// TwinCAT 3 PLC project PLCIO
// ProgramVersion: 3.1.4026.10
// libraries:
//   Tc2_ControllerToolbox, * (Beckhoff Automation GmbH)
//   Tc2_IoFunctions, * (Beckhoff Automation GmbH)
//   Tc2_ModbusRTU, * (Beckhoff Automation GmbH)
//   Tc2_ModbusSrv, * (Beckhoff Automation GmbH)
//   Tc2_SerialCom, * (Beckhoff Automation GmbH)
//   Tc2_Standard, * (Beckhoff Automation GmbH)
//   Tc2_System, * (Beckhoff Automation GmbH)
//   Tc2_Utilities, * (Beckhoff Automation GmbH)
//   Tc3_BA_Common, * (Beckhoff Automation GmbH)
//   Tc3_EventLogger, * (Beckhoff Automation GmbH)
//   Tc3_Module, * (Beckhoff Automation GmbH)
// project tree:
//   / CheckDivDInt.TcPOU, CheckDivLInt.TcPOU (not stored), CheckDivLReal.TcPOU, CheckDivReal.TcPOU (not stored), PlcTask.TcTTO (not stored), PlcTask_Fast.TcTTO (not stored)
//   DUTs/ outWord.TcDUT, ScaleFactor.TcDUT, ST_Device.TcDUT, RecipeStep.TcDUT
//   FUNTION/ BOOL_TO_STRING_LHeaterON.TcPOU, CheckRangeSigned.TcPOU (not stored), CheckRangeUnsigned.TcPOU (not stored), HEXSTR_TO_REAL_LHeaterPV.TcPOU, Real_To_String_LineHeater.TcPOU, Real_To_String_ThermalBath.TcPOU, USINT_TO_WORD_Bit.TcPOU, WORD_TO_USINT_Bit.TcPOU (not stored)
//   GVLs/ GVL.TcGVL (not stored), GVL_Interlock.TcGVL, GVL_Serial.TcGVL (not stored), GVL_IO.TcGVL, RCP.TcGVL (not stored)
//   POUs/ FB_RecipeSequencer.TcPOU (not stored), backup2.TcPOU (not stored), backup1.TcPOU, Test_Recipe_Run.TcPOU, FB_RampGeneration_Gas.TcPOU (not stored), MAIN.TcPOU (not stored), P11_E3508.TcPOU, P12_IQ_PLUS.TcPOU, P13_LineHeater.TcPOU, P14_ThermalBath.TcPOU (not stored), P15_RotationOperation.TcPOU (not stored), P16_CoverOperation.TcPOU (not stored), P17_DOROperation.TcPOU (not stored), P20_BackgroundCom.TcPOU, P21_Background_LineHeater.TcPOU (not stored), P22_Background_ThermalBath.TcPOU (not stored), P50_RecipeControl.TcPOU (not stored), P90_Interlock.TcPOU (not stored), P91_Monitoring.TcPOU (not stored), P92_Maintenance.TcPOU (not stored), P93_Setting.TcPOU (not stored)

// ---- DUTs/outWord.TcDUT
TYPE outWord :
STRUCT
	Lower : USINT; //Lower Bytes
	Upper : USINT; //Upper Bytes
END_STRUCT
END_TYPE

// ---- DUTs/ScaleFactor.TcDUT
TYPE ScaleFactor :
STRUCT
	MinFactor	: USINT; // Sensor Minimum Range
	MaxFactor	: USINT; // Sensor Maximum Range
END_STRUCT
END_TYPE

// ---- DUTs/ST_Device.TcDUT
TYPE ST_Device :
STRUCT
	aDigitalInputIO  	: ARRAY[1..9]OF BYTE; //KL1408 9EA
	aDigitalOutputIO  	: ARRAY[1..4]OF BYTE; //KL2408 4EA
	
	// Analog Input to INT
	aAnalogInputIO 		: ARRAY[1..40]OF INT;
	aAnalogOutputIO 	: ARRAY[1..28]OF INT;
	aAnalogInputIO2 	: ARRAY[1..2]OF UINT;
	//Solenoid Valve
	aOutputSolValve  	: ARRAY[1..2]OF DWORD; //Solenoid Valve 
END_STRUCT
END_TYPE

// ---- DUTs/RecipeStep.TcDUT
TYPE RecipeStep :
STRUCT
	iRecipe : ARRAY[1..9] OF INT; //Reactor Condition
	rRecipe : ARRAY[1..26] OF REAL; //MFC, EPC Data
	dRecipe : DWORD; //Valve Data
	sRecipe : STRING(81);
END_STRUCT
END_TYPE

// ---- GVLs/GVL_Interlock.TcGVL
{attribute 'qualified_only'}
VAR_GLOBAL
	
END_VAR

// ---- GVLs/GVL_IO.TcGVL
{attribute 'qualified_only'}
VAR_GLOBAL
	// Digital IO to Byte
	aDigitalInputIO AT %I* 	: ARRAY[1..9]OF BYTE; //KL1408 9EA
	aDigitalOutputIO AT %Q* : ARRAY[1..4]OF BYTE; //KL2408 4EA

	// Analog Input to INT
	aAnalogInputIO AT %I* 	: ARRAY[1..40]OF INT;
	aAnalogOutputIO AT %Q* 	: ARRAY[1..28]OF INT;
	aAnalogInputIO2 AT %I*	: ARRAY[1..2]OF UINT;
	//Solenoid Valve
	aOutputSolValve AT %Q* 	: ARRAY[1..2]OF DWORD; //Solenoid Valve 
	// Variable(struct) Connecting PC to PLC 
	stDeviceIO				: ST_Device;

	aMaxValue	: ARRAY[1..50]OF REAL; //Device Max Value from UI
	
	
END_VAR

// ---- CheckDivDInt.TcPOU
// Implicitly generated code : DO NOT EDIT
FUNCTION CheckDivDInt : DINT
VAR_INPUT
	divisor:DINT;
END_VAR

// Implicitly generated code: Only an implementation suggestion
{noflow}
IF divisor = 0 THEN
	CheckDivDInt:=1;
ELSE
	CheckDivDInt:=divisor;
END_IF;

END_FUNCTION

// ---- CheckDivLReal.TcPOU
// Implicitly generated code : DO NOT EDIT
FUNCTION CheckDivLReal : LREAL
VAR_INPUT
	divisor:LREAL;
END_VAR

// Implicitly generated code: Only an implementation suggestion
{noflow}
IF divisor = 0 THEN
	CheckDivLReal:=1;
ELSE
	CheckDivLReal:=divisor;
END_IF;

END_FUNCTION

// ---- FUNTION/BOOL_TO_STRING_LHeaterON.TcPOU
FUNCTION BOOL_TO_STRING_LHeaterON : STRING
VAR_INPUT
	nHeaterNumber	: INT;
	bON				: BOOL;
END_VAR
VAR
	sString			: STRING;
	sHeaterNumber	: STRING;
END_VAR

//LH: Line Heater x 8EA -> 8Channel TIC 1EA
//Model: HANYOUNG NUX, MC9-8RD0SS32

//STRING : '$0201DWR,02,0302(CH_NO),0001(CH_1),0501(AT),0001(AT-ON)
sString := '$0201DWR,02,0302,,0501,000$0D$0A';

//Convert to Channel from Heater Number
sHeaterNumber := DINT_TO_DECSTR(nHeaterNumber, 4);
sString := INSERT(sString,sHeaterNumber,15);

IF bON = TRUE THEN
	sString := INSERT(sString,'1',28);
ELSE
	sString := INSERT(sString,'0',28);
END_IF

BOOL_TO_STRING_LHeaterON := sString;

END_FUNCTION

// ---- FUNTION/HEXSTR_TO_REAL_LHeaterPV.TcPOU
FUNCTION HEXSTR_TO_REAL_LHeaterPV : REAL
VAR_INPUT
	hStrTemperaturePV : STRING;
END_VAR
VAR
	hData			:UDINT;
	aData	: ARRAY[0..1]OF BYTE;
	bSwap	: BYTE;
	ptStrTemperature : POINTER TO INT;
	nTemperaturePV : INT;
END_VAR

// Convert to Data Array from HexString
hData := HEXSTR_TO_DATA(hStrTemperaturePV, ADR(aData), SIZEOF(aData));

//Swap Data
bSwap := aData[0];
aData[0] := aData[1];
aData[1] := bSwap;

ptStrTemperature := ADR(aData);
nTemperaturePV := ptStrTemperature^;
HEXSTR_TO_REAL_LHeaterPV := INT_TO_REAL(nTemperaturePV);

END_FUNCTION

// ---- FUNTION/Real_To_String_LineHeater.TcPOU
FUNCTION Real_To_String_LineHeater : STRING
VAR_INPUT
	rTemperatureSV 		: REAL;
	nHeaterNumber		: INT;
END_VAR
VAR
	wTemperature		: WORD;
	hStrTemp			: STRING;
	sHeaterNumber		: STRING;
	sString				: STRING;
	sSendString			: STRING;
END_VAR

//LH: Line Heater x 8EA -> 8Channel TIC 1EA
//Model: HANYOUNG NUX, MC9-8RD0SS32

// Multiple decimal place point
// STRING : '$0201DWR,03,0301(ZONE_NO),0001(ZONE_1),0302(CH_NO),0001(CH_1,sHeaterNumber),0401(SV), hStrTemp, $0D$0A'
sString := '$0201DWR,03,0301,0001,0302,,0401,,$0D$0A';

//Convert to Channel from Heater Number
sHeaterNumber := DINT_TO_DECSTR(nHeaterNumber, 4);
sString := INSERT(sString,sHeaterNumber,25);
	
//Convert to String Type
wTemperature := REAL_TO_WORD(rTemperatureSV);
hStrTemp := WORD_TO_HEXSTR(wTemperature, 4, FALSE);
Real_To_String_LineHeater := INSERT(sString,hStrTemp,35);

END_FUNCTION

// ---- FUNTION/Real_To_String_ThermalBath.TcPOU
FUNCTION Real_To_String_ThermalBath : STRING
VAR_INPUT
	rTemperatureSV 	: REAL;
	nBathNumber		: INT;
END_VAR
VAR
	sBathNumber 	: STRING;
	rTemp 			: REAL;
	nTemp 			: DINT;
	sTemp 			: STRING;
	sBaseString		: STRING;
END_VAR

// Thermal Bath SMC HEBC002-WA10
rTemp := rTemperatureSV*10 ;
nTemp := REAL_TO_DINT(rTemp);
sBaseString := '$020WSV1$03';

sBathNumber := INT_TO_STRING(nBathNumber);
sBaseString := INSERT(sBaseString,sBathNumber,2);

IF nTemp >= 0 THEN
	sTemp := DINT_TO_DECSTR(nTemp, 5); //00010
ELSE
	sTemp := DINT_TO_DECSTR(nTemp, 4); 
	sTemp := CONCAT('-',sTemp); //-0010
END_IF

sBaseString := INSERT(sBaseString,sTemp,7);

Real_To_String_ThermalBath := sBaseString;

END_FUNCTION

// ---- FUNTION/USINT_TO_WORD_Bit.TcPOU
//2-USINT combine to 1-WORD converting using a bit operation
FUNCTION USINT_TO_WORD_Bit : WORD
VAR_INPUT
	aInput_L : USINT; //Lower
	aInput_U : USINT; //Upper
END_VAR
VAR
	nWord_L : WORD; //Lower
	nWord_U : WORD; //Upper
END_VAR

nWord_L := TO_WORD(aInput_L);
// 1111_1111
// 0000_0000_1111_1111
nWord_U := TO_WORD(aInput_U);
// 1111_1111
// 0000_0000_1111_1111
nWord_U := SHL(nWord_U, 8);
// 1111_1111_0000_0000
USINT_TO_WORD_Bit := TO_WORD(nWord_L OR nWord_U);

END_FUNCTION

// ---- POUs/backup1.TcPOU
PROGRAM P50_RecipeControl1
VAR
	RcpIndex	: INT;
	
	iTimerCount: INT;
	OnTimer: TON;
	OffTimerOut: BOOL;
	OnTimerOut: BOOL;
	timeTrigOn: R_TRIG;
	
	bTrigOn: BOOL;
	ReverseSignal: BOOL;
	OffTimer: TOF;
	fb_RecipeSequencer : FB_RecipeSequencer;
END_VAR

IF RCP.bRcpInit THEN
	(* reset the init flag *)
	iTimerCount := 0;
	RcpIndex := 1;
	RCP.bRcpInit := FALSE;
END_IF

IF RcpIndex <= RCP.iRcpTotalStep THEN
	OnTimer(IN:=OffTimerOut, Pt:= INT_TO_TIME(500), Q=>OnTimerOut, ET=>);
	timeTrigOn(clk:=OnTimerout, Q=>bTrigOn);
	IF (bTrigOn AND RCP.iRcpOperationState) THEN
		iTimerCount := iTimerCount +1;
		bTrigOn := FALSE;
		
		IF iTimerCount <= RCP.aRecipe[RcpIndex].iRecipe[2] THEN
			fb_RecipeSequencer(nRcpIndex:=RcpIndex);
			
		ELSIF iTimerCount > RCP.aRecipe[RcpIndex].iRecipe[2] + RCP.aRecipe[RcpIndex].iRecipe[3] THEN
			iTimerCount := 0;
			RcpIndex := RcpIndex + 1;
		END_IF
	END_IF
	IF OnTimerOut = TRUE THEN
		ReverseSignal := FALSE;
	ELSE
		ReverseSignal := TRUE;
	END_IF

	OffTimer(in:=ReverseSignal, pt:= INT_TO_TIME(500), q=>OffTimerOut,et=>);
END_IF

END_PROGRAM

// ---- POUs/Test_Recipe_Run.TcPOU
PROGRAM Test_Recipe_Run
VAR
// 	fb_RecipeSequencer : FB_RecipeSequencer;
	bMaintKey : BOOL;
	bPc2Plc	: BOOL;
	
	plc_state	: BOOL;
	plc_array	: BYTE;
	
	iRcpCurrNum : INT := 1;
	iTimerCount	: INT;

	timeTrigOn	: r_trig;
	bTrigOn		: BOOL;
	bRcpInit	: BOOL;
	bRcpEnable	: BOOL;
	fb_RecipeSequencer : FB_RecipeSequencer;

	ctime : TIME :=  T#1D14H30M40S500MS;
	lctime : LTIME ;
	
	cdate : DATE :=  D#2024-07-07;
	str : STRING ;
	wstr : STRING;
	tempstr : STRING;

	OnTimer : TON;
	OffTimer : TOF;
	EnableTimer : BOOL;
	TimerOutPut : BOOL;	
	OnTimerOut : BOOL := FALSE;
	ReverseSignal : BOOL;
	OffTimerOut : BOOL;
	count : INT;
	el2088_out : BYTE;
	el4024_out : INT;
	el3054_in : INT;
	
END_VAR

// Load current recipe of recipes array 
bMaintKey := GVL_IO.aDigitalInputIO[1].0;

// Connect PLC varibaes to PC variables
IF bPc2Plc = TRUE THEN
	GVL_IO.aDigitalInputIO := GVL_IO.stDeviceIO.aDigitalInputIO;
	GVL_IO.aDigitalOutputIO := GVL_IO.stDeviceIO.aDigitalOutputIO;
	GVL_IO.aAnalogInputIO := GVL_IO.stDeviceIO.aAnalogInputIO;
	GVL_IO.aAnalogOutputIO := GVL_IO.stDeviceIO.aAnalogOutputIO;
	GVL_IO.aAnalogInputIO2 := GVL_IO.stDeviceIO.aAnalogInputIO2;
	GVL_IO.aOutputSolValve := GVL_IO.stDeviceIO.aOutputSolValve;
	bPc2Plc := FALSE;
ELSE
	GVL_IO.stDeviceIO.aDigitalInputIO  := GVL_IO.aDigitalInputIO; 
	GVL_IO.stDeviceIO.aDigitalOutputIO := GVL_IO.aDigitalOutputIO;
	GVL_IO.stDeviceIO.aAnalogInputIO   := GVL_IO.aAnalogInputIO;
	GVL_IO.stDeviceIO.aAnalogOutputIO  := GVL_IO.aAnalogOutputIO; 
	GVL_IO.stDeviceIO.aAnalogInputIO2  := GVL_IO.aAnalogInputIO2; 
	GVL_IO.stDeviceIO.aOutputSolValve  := GVL_IO.aOutputSolValve;
END_IF

IF bRcpInit THEN
	(* reset the init flag *)
	iTimerCount := 0;
	iRcpCurrNum := 1;
	bRcpInit := FALSE;
END_IF

IF iRcpCurrNum <= 50 THEN
	OnTimer(IN:=OffTimerOut, Pt:= INT_TO_TIME(500), Q=>OnTimerOut, ET=>);
	timeTrigOn(clk:=OnTimerout, Q=>bTrigOn);
	IF (bTrigOn AND GVL.bRunRecipe) THEN
		iTimerCount := iTimerCount +1;
		bTrigOn := FALSE;
		
		IF iTimerCount <= RCP.aRecipe[iRcpCurrNum].iRecipe[2] THEN
			fb_RecipeSequencer(nRcpIndex:=iRcpCurrNum);
			
		ELSIF iTimerCount > RCP.aRecipe[iRcpCurrNum].iRecipe[2] + RCP.aRecipe[iRcpCurrNum].iRecipe[3] THEN
			iTimerCount := 0;
			iRcpCurrNum := iRcpCurrNum + 1;
		END_IF
	END_IF
	IF OnTimerOut = TRUE THEN
		ReverseSignal := FALSE;
	ELSE
		ReverseSignal := TRUE;
	END_IF

	OffTimer(in:=ReverseSignal, pt:= INT_TO_TIME(500), q=>OffTimerOut,et=>);
END_IF


cdate :=  D#2024-07-07;
str := 'We are the one, let us heading forwards';

count := count + 1;

GVL.EL4024_OUT := el4024_out;
el3054_in := GVL.EL3054_IN;

plc_array := EL2088_OUT;

END_PROGRAM

// ---- POUs/P11_E3508.TcPOU
PROGRAM P11_E3508
VAR_INPUT
	nTemperatureTargetValue	: INT(0..1200); //Target Values, Input Range 0 ~ 1200 Celcius
	nRampTime				: INT := 1; //Second
	nPowerRateSetValue		: WORD;	
	bOutputManAuto 			: BOOL; // 0:Auto, 1:Manual Operation
	
	bHeaterOn				: BOOL := FALSE; //to PSTEK
	bHeaterReset			: BOOL; //to PSTEK

END_VAR
VAR_OUTPUT
	bAlarmState_E3508 		: BOOL; //Alarm or Sensor Break Signal
	bManAuto_E3508 			: BOOL; // 0:Manual, 1:Auto
	rPowerRate				: REAL;	//Power rate for Monitoring
	
	isHeaterReady			: BOOL; //Close : Ready
	isHeaterRun				: BOOL; //Close : Running, Open : Stop
	isHeaterFault			: BOOL; //Close : Falut, Open : Normal
	//isInductionHeaterErr	: BOOL; //Power Supply
	bInductionHeaterCB		: BOOL;
END_VAR

VAR
	//Input from E3508 Controller
	aInputPVBytes AT %I* 		: ARRAY[1..2]OF USINT; //Input Process Values
	aInputSVBytes AT %I* 		: ARRAY[1..2]OF USINT; //Input Set Values
	aInputTVBytes AT %I* 		: ARRAY[1..2]OF USINT; //Input Target Valuse
	aInputCVBytes AT %I* 		: ARRAY[1..2]OF USINT; //Induction Heter Controlled Values
	aInputProportional AT %I* 	: ARRAY[1..2]OF USINT; //PID - Proportional Band
	aInputIntegral AT %I* 		: ARRAY[1..2]OF USINT; //PID - Integral Time
	aInputDerivative AT %I* 	: ARRAY[1..2]OF USINT; //PID - Derivative Time 
	nInputAlarmBytes AT %I* 	: USINT; // Alarm State
	nInputManAutoBytes AT %I* 	: USINT; // ManAuto State
	
	nTemperaturePV_E3508		: WORD;
	nTemperatureSV_E3508		: WORD;
	nPowerRate_E3508		: WORD; //To Induction Heater Control Values
	nParameterP				: WORD; //PID Parameter P
	nParameterI				: WORD; //PID Parameter I
	nParameterD				: WORD; //PID Parameter D
	//Output to E3508 Controller
	wOutputSVBytes 				: outWord;
	wOutputPowerSVBytes 		: outWord;
	aOutputSVBytes AT %Q* 		: ARRAY[1..2]OF USINT; //Temperature Set Value
	nOutputManAutoBytes AT %Q* 	: USINT; //ManAuto Change
	aOutputPowerBytes AT %Q* 	: ARRAY[1..2]OF USINT; //Output Power in Manual State
	//nOutputAlarmClear AT %Q* : USINT; //Alarm Clear Set
	
	nTemperatureControlValue	: WORD;
	
	// for FB_CTRL_RAMP_GENERATOR Variable
	(* input *)
	bEnable					: BOOL;
	rTemperatureStartValue	: REAL;
	rTemperatureTargetValue	: REAL;
	(* output *)
	rTemperatureControlValue : LREAL;
	bValueReached			: BOOL;
	(* function block *)
	fbCTRL_RAMP_GENERATOR		: FB_CTRL_RAMP_GENERATOR;
	stCTRL_RAMP_GENERATOR_PARAMS: ST_CTRL_RAMP_GENERATOR_PARAMS;

	eErrorId				: E_CTRL_ERRORCODES;
	bError					: BOOL;
	bInit					: BOOL := TRUE;

	(* Induction Heating Operation Parameter*)
	rRampingRatio			: REAL;	
END_VAR

//Induction Heater & Temperature Controller & Thermo Couple(R-Type)
//Maker: PSTEK, Eurotherm
//Model: 3508
//Temperature Range: 0 ~ 12000℃

(* Read from Power Distribution Pannel *)
bInductionHeaterCB		:= GVL_IO.aDigitalInputIO[4].7;

(* Read from E3508 Device Value *)
nTemperaturePV_E3508	:= USINT_TO_WORD_Bit(aInputPVBytes[1], aInputPVBytes[2]);
nTemperatureSV_E3508	:= USINT_TO_WORD_Bit(aInputSVBytes[1], aInputSVBytes[2]);
nPowerRate_E3508		:= USINT_TO_WORD_Bit(aInputCVBytes[1], aInputCVBytes[2]); //divided to 10
nParameterP 			:= USINT_TO_WORD_Bit(aInputProportional[1], aInputProportional[2]);
nParameterI 			:= USINT_TO_WORD_Bit(aInputIntegral[1], aInputIntegral[2]);
nParameterD 			:= USINT_TO_WORD_Bit(aInputDerivative[1], aInputDerivative[2]);

bAlarmState_E3508 		:= nInputAlarmBytes.7;
bManAuto_E3508 			:= nInputManAutoBytes.7;

(* Read from Induction Heater Value *)
isHeaterReady 			:= GVL_IO.aDigitalInputIO[2].2;
isHeaterRun		 		:= GVL_IO.aDigitalInputIO[2].3;
isHeaterFault 			:= GVL_IO.aDigitalInputIO[2].4;

(*Ramp Generator Parameter Variable*)
rTemperatureTargetValue	:= INT_TO_REAL(nTemperatureTargetValue);
rPowerRate				:= WORD_TO_REAL(nPowerRate_E3508)*0.1; //divided to 10

bHeaterOn := TRUE;
bInit := NOT((rTemperatureTargetValue = 0) AND (rTemperatureStartValue = 0));

IF bInit AND nRampTime <> 0 AND RCP.iRcpOperationState=10 THEN
	rRampingRatio := ABS(rTemperatureTargetValue - rTemperatureStartValue) / nRampTime; //Second
	(* init parameter struct *)
	stCTRL_RAMP_GENERATOR_PARAMS.tTaskCycleTime		:= T#2MS;
	stCTRL_RAMP_GENERATOR_PARAMS.tCtrlCycleTime		:= T#100MS;
	stCTRL_RAMP_GENERATOR_PARAMS.fVeloPos			:= rRampingRatio; (* in units per second *)
	stCTRL_RAMP_GENERATOR_PARAMS.fVeloNeg			:= rRampingRatio; (* in units per second *)

	IF rTemperatureTargetValue <> rTemperatureStartValue THEN
		bEnable := TRUE;
		(* call function block *)
		fbCTRL_RAMP_GENERATOR(
			bEnable			:= bEnable,
			fStart			:= rTemperatureStartValue,
			fTarget			:= rTemperatureTargetValue,
			stParams		:= stCTRL_RAMP_GENERATOR_PARAMS,
			fOut			=> rTemperatureControlValue,
			bValueReached	=> bValueReached,
			bError			=> bError,
			eErrorId		=> eErrorId);
	ELSE
		fbCTRL_RAMP_GENERATOR.bEnable := FALSE;
	END_IF

	IF bValueReached THEN
		rTemperatureStartValue	:= LREAL_TO_REAL(rTemperatureControlValue);
	END_IF
END_IF

nTemperatureControlValue	:= LREAL_TO_WORD(rTemperatureControlValue);

(* Write to E3508 Device Value *)
wOutputSVBytes 			:= WORD_TO_USINT_Bit(nTemperatureControlValue);
aOutputSVBytes[1] 		:= wOutputSVBytes.Lower;
aOutputSVBytes[2] 		:= wOutputSVBytes.Upper;

// PowerRate Operation
nOutputManAutoBytes.0 	:= bOutputManAuto;

wOutputPowerSVBytes 	:= WORD_TO_USINT_Bit(nPowerRateSetValue*10); //multiple to 10
aOutputPowerBytes[1] 	:= wOutputPowerSVBytes.Lower;
aOutputPowerBytes[2] 	:= wOutputPowerSVBytes.Upper;

(* Write to Induction Heater Value *)
GVL_IO.aDigitalOutputIO[2].0 := bHeaterOn;
GVL_IO.aDigitalOutputIO[2].1 := bHeaterReset;

END_PROGRAM

// ---- POUs/P12_IQ_PLUS.TcPOU
PROGRAM P12_IQ_PLUS
VAR_INPUT
	nPressureTargetValue : WORD := 760;//Pressure Set Value
	nRampTime			: INT := 1; //Second
	//wSetPoint 			: WORD; //Set Point
	nSetType 			: USINT; //1:Pressure Conrol, 2:Position Control
	nTValveMode 		: USINT := 0; //Valve Mode
	bPumpOn				: BOOL;
	bPumpReset			: BOOL;
	
	bEnable				: BOOL; //Value Change

END_VAR
VAR_OUTPUT
	rPressurePV_CD1 	: REAL; //CD2 Current Pressure
	rPressurePV_CD2 	: REAL; //CD2 Current Pressure
	rValvePosition 		: REAL; //Valve Position
	bVacuumPumpCB		: BOOL;
	bThrottleValveCP	: BOOL;
	nPressureControlValue	: INT;

	//nInputStatus
	ingPressureControl 	: BOOL;
	ingPositionControl 	: BOOL;
	isValveOpen 			: BOOL;
	isValveNotInitialized 	: BOOL;	
	isValveClosed 			: BOOL;
	isValveFaultState 		: BOOL;
	ingValveInitializing 	: BOOL;
	ingHoldState 			: BOOL;
	
	// Vacuum Pump Status
	isPumpFault				: BOOL;
	isPumpWarning			: BOOL;
	isPumpAlarm				: BOOL;
	isFBRunning				: BOOL;
	isPumpRunning			: BOOL;
	
END_VAR
VAR
	//Input from IQ-PLUS Throttle Valve
	nInputStatus AT %I* : USINT; //Input Status Bytes
	aInputPressurePV_CDG1 AT %I* : ARRAY[1..2]OF USINT; //CDG1 Pressure
	aInputPressurePV_CDG2 AT %I* : ARRAY[1..2]OF USINT; //CDG2 Pressure
	aInputPressureSP AT %I* : ARRAY[1..2]OF USINT; //Set Point Pressure
	aInputValvePosionPV AT %I* : ARRAY[1..2]OF USINT; //Current Valve Position
	
	wOutputSetPoint : WORD;
	oSetPoint : outWord; //Word to Byte variable
	
	//Output to IQ-PLUS Throttle Valve
	nOutputMode AT %Q* : USINT;
	aOutputSPBytes AT %Q* : ARRAY[1..2]OF USINT; //Set Pressure
	nOutputSetType AT %Q* : USINT; //1:Pressure Control, 2:Valve Position Control
	wInputPressurePV_CDG1 : WORD; //CDG1 Current Pressure, Not Used
	wInputPressurePV_CDG2 : WORD; //CDG2 Current Pressure
	wInputValvePosition : WORD; //Current Valve Position (0~100%)
	nInputStatusOld : USINT := 9; //Value Change Monitoring, First Temp value
	
	// for FB_CTRL_RAMP_GENERATOR Variable
	(* input *)
	rPressureTargetValue 		: REAL;
	rPressureStartValue 		: REAL := 760;
	(* output *)
	rPressureControlValue		: LREAL;
	bValueReached				: BOOL;
	(* function block *)
	fbCTRL_RAMP_GENERATOR			: FB_CTRL_RAMP_GENERATOR;
	stCTRL_RAMP_GENERATOR_PARAMS	: ST_CTRL_RAMP_GENERATOR_PARAMS;
	eErrorId						: E_CTRL_ERRORCODES;
	bError							: BOOL;
	bInit						: BOOL := TRUE;	
	(* Operation Parameter*)
	rRampingRatio				: REAL;	
	rPressureControlValue_torr	: lreal;
END_VAR
VAR CONSTANT
	//Conversion Parameter
	SetPointFactor : REAL := 327.67; //Range 0~7FFFh
	PressureFactor : REAL := 24.576;	//Range 0~6000h
END_VAR

//Model : IQ Plus 
//Pressure Range : 0 ~ 1,000 Torr

(* Read from Power Distribution Pannel *)
bVacuumPumpCB		:= GVL_IO.aDigitalInputIO[5].1;
bThrottleValveCP 	:= GVL_IO.aDigitalInputIO[5].5; //Throttle Valve CP

(* Read from Vacuum Pump *)
isPumpFault			:= GVL_IO.aDigitalInputIO[2].7;
isPumpWarning		:= GVL_IO.aDigitalInputIO[3].0;
isPumpAlarm			:= GVL_IO.aDigitalInputIO[3].1;
isFBRunning			:= GVL_IO.aDigitalInputIO[3].2;
isPumpRunning		:= GVL_IO.aDigitalInputIO[3].3;

(* Read from Device Value *)
// 2USINT to WORD
wInputPressurePV_CDG1 	:= USINT_TO_WORD_Bit(aInputPressurePV_CDG1[1],aInputPressurePV_CDG1[2]);
wInputPressurePV_CDG2 	:= USINT_TO_WORD_Bit(aInputPressurePV_CDG2[1],aInputPressurePV_CDG2[2]);
wInputValvePosition 	:= USINT_TO_WORD_Bit(aInputValvePosionPV[1], aInputValvePosionPV[2]);

//From IQ Plus
rPressurePV_CD1 := WORD_TO_REAL(wInputPressurePV_CDG1)/PressureFactor;
rPressurePV_CD2 := WORD_TO_REAL(wInputPressurePV_CDG2)/PressureFactor;
rValvePosition := WORD_TO_REAL(wInputValvePosition)/SetPointFactor;

nSetType := 1;
//To IQ Plus
IF nTValveMode = 0 AND nSetType = 1 THEN
	rPressureTargetValue := nPressureTargetValue * SetPointFactor * 0.1; //Pressure Control
ELSIF nTValveMode = 0 AND nSetType = 2 THEN
	rPressureTargetValue := nPressureTargetValue * SetPointFactor; // Position Control
END_IF

//Ramp Generator
bInit := NOT((rPressureTargetValue = 0) AND (rPressureStartValue = 0));

IF bInit AND nRampTime <> 0 AND RCP.iRcpOperationState=10 THEN
	rRampingRatio := ABS(rPressureTargetValue - rPressureStartValue) / nRampTime; // Second
	(* init parameter struct *)
	stCTRL_RAMP_GENERATOR_PARAMS.tTaskCycleTime		:= T#2MS;
	stCTRL_RAMP_GENERATOR_PARAMS.tCtrlCycleTime		:= T#100MS;
	stCTRL_RAMP_GENERATOR_PARAMS.fVeloPos			:= rRampingRatio; (* in units per second *)
	stCTRL_RAMP_GENERATOR_PARAMS.fVeloNeg			:= rRampingRatio; (* in units per second *)
	(* reset the init flag *)
	bInit := FALSE;

	IF rPressureTargetValue <> rPressureStartValue THEN
		bEnable := TRUE;
		(* call function block *)
		fbCTRL_RAMP_GENERATOR(
			bEnable			:= bEnable,
			fStart			:= rPressureStartValue,
			fTarget			:= rPressureTargetValue,
			stParams		:= stCTRL_RAMP_GENERATOR_PARAMS,
			fOut			=> rPressureControlValue,
			bValueReached	=> bValueReached,
			bError			=> bError,
			eErrorId		=> eErrorId);
	ELSE
		fbCTRL_RAMP_GENERATOR.bEnable := FALSE;
	END_IF

	IF bValueReached THEN
		rPressureStartValue := LREAL_TO_REAL(rPressureControlValue);
	END_IF
END_IF


wOutputSetPoint := LREAL_TO_WORD(rPressureControlValue);
oSetPoint := WORD_TO_USINT_Bit(wOutputSetPoint);
aOutputSPBytes[1] := oSetPoint.Lower;
aOutputSPBytes[2] := oSetPoint.Upper;

nOutputSetType := nSetType;

//Valve Status Initailize
IF nInputStatus <> nInputStatusOld THEN
	// Staus Initializing
	ingPressureControl := FALSE;
	ingPositionControl := FALSE;
	isValveOpen := FALSE;
	isValveNotInitialized := FALSE;	
	isValveClosed := FALSE;
	isValveFaultState := FALSE;
	ingValveInitializing := FALSE;
	ingHoldState := FALSE;
	// Status Update	
	nInputStatusOld := nInputStatus;
END_IF

//Update Valve Status
CASE nInputStatus OF
	0 : ingPressureControl := TRUE; //Pressure Control Performing.
	1 : ingPositionControl := TRUE; //Position Control Performing.	
	2 : isValveOpen := TRUE; //Valve Open, Stopped, Not Controlling.
	3 : isValveNotInitialized := TRUE; //Valve not initialized power on or RESET Command.
	4 : isValveClosed := TRUE; //Valve Closed, Stopped, Not Controlling.
	5 : isValveFaultState := TRUE; //Has faulted during valve initialization or operation.
	6 : ingValveInitializing := TRUE; //Initailizing Process.
	8 : ingHoldState := TRUE; //intermediate position, not at open or close and not controlling pressure.
END_CASE

// nOutputMode
// 0 : uses setpoint and setpoint type to control the valve.
// 1 : Does not use setpoint and setpoint type to operate the valve.
// 2 : Does not use setpoint and setpoint type to operate the valve.
// 3 : Holds valve in current position.
// 4 : Reset the controller.
nOutputMode := nTValveMode;
nPressureControlValue := LREAL_TO_INT(rPressureControlValue);

rPressureControlValue_torr := LREAL_TO_REAL(rPressureControlValue / SetPointFactor * 10);

 //Pressure Control

GVL_IO.aDigitalOutputIO[2].2 := bPumpOn; //Pump On
GVL_IO.aDigitalOutputIO[2].3 := bPumpReset; // Pump Reset

END_PROGRAM

// ---- POUs/P13_LineHeater.TcPOU
PROGRAM P13_LineHeater
VAR_INPUT
	rTemperatureSV 		: ARRAY[1..8]OF REAL;
	bAutoTuneSV 		: ARRAY[1..8]OF BOOL;
END_VAR
VAR_OUTPUT
	rTemperaturePV 		: ARRAY[1..8]OF REAL;
	isLineHeater_Run	: ARRAY[1..8]OF BOOL;
	isLineHeater_ATune	: ARRAY[1..8]OF BOOL;
	isLineHeater_Err	: ARRAY[1..8]OF BOOL;
END_VAR
VAR
	TimeOnDelay			: TON; //Time delay after Power ON of Thermal Bath
	TimeCycle			: TON;
	nComMode 			: INT; // //1 = PV Req, 2 = STATUS Req, 3 = SV Write, 4 = AutoTune On/Off
	nCount 				: INT;
	rTemperatureTV 		: ARRAY[1..8]OF REAL;
	bAutoTuneTV			: ARRAY[1..8]OF BOOL;

	//for sending variable
	TimeWaitSend		: TON;
	bSendingEnable 		: BOOL:=TRUE; // Check the Sending Stage
	bSetValueMode 		: BOOL;
	fbSend				: SendString;
	sSendString 		: STRING;
	bSendBusy			: BOOL;
	bSendingOK 			: BOOL; //v1
	eSendErrorID		: ComError_t;
	
	// for received variable
	TimeWaitReceive		:TON;
	fbReceive			: ReceiveString;
	sReceivedString		: STRING;
	bStringReceived		: BOOL;
	bReceiveBusy		: BOOL;
	bReceiveError		: BOOL;
	eReceiveErrorID		: ComError_t;
	bReceiveTimeout		: BOOL;
	bReceivedOK 		: BOOL;
	hStrReceivedST		: STRING;
	hStrReceivedPV		: STRING;
	
	nHeaterNumber 		: INT := 1;
	sHeaterNumber 		: STRING := '1';
	sReceivedHeaterNumber : STRING;
	nReceivedHeaterNumber : INT;
	sReceivedAffirmation : STRING;
	sReceivedData 		: STRING;
	nHeaterStrPositionPV : INT:= 11; //Received String Start Position
	nDecimal			:INT;
	nSendStrCounter		:INT := 1;
	bReset : BOOL;
	sTest : STRING;
	nStrPosition : INT;
	nHeaterNumberPV : INT;
	sTemperaturePV : STRING;
	(* Input *)
	bLineHeaterCB		: BOOL;
	bLineHeaterCP		: BYTE;
END_VAR

//LH: Line Heater x 8EA -> 8Channel TIC 1EA
//Maker: HANYOUNG NUX
//Model: MC9-8RD0SS32
//Temp Range: -15 ~200℃
//RS485: 9600, DataBit(8), Parity(None), StopBit(1)
//BCC Check X

(* Read from Device Value *)
// Line Heater CP
bLineHeaterCB	:= GVL_IO.aDigitalInputIO[5].2;
bLineHeaterCP 	:= GVL_IO.aDigitalInputIO[6]; //LineHeaterCP1   := bLineHeaterCP.0, Until CP8

// make a sending string
TimeOnDelay(IN:= P90_Interlock.bLineHeaterMC, PT :=T#5S); //Time Delay after a Thermal Bath MC ON
IF TimeOnDelay.Q THEN
	TimeOnDelay(IN:=FALSE);
	// Make a sending string Set value or Request value 
	IF bSendingEnable = FALSE THEN
		bSendingEnable := TRUE;
		bSendingOK := FALSE;
		bReceivedOK := FALSE;
		
		IF nComMode <>1 THEN
			sSendString := '$0201DRS,08,0001$0D$0A'; //Request PV
			nComMode := 1;
		ELSE
			sSendString := '$0201DRS,08,0111$0D$0A'; //Request State
			nComMode := 2;
		END_IF
	
		FOR nHeaterNumber:= 1 TO 8 DO
			IF (rTemperatureTV[nHeaterNumber] <> rTemperatureSV[nHeaterNumber]) THEN
				// if SetValue are different to TargetValue, change Target vale to setvalue
				rTemperatureTV[nHeaterNumber] := rTemperatureSV[nHeaterNumber];
				sSendString := Real_To_String_LineHeater(rTemperatureTV[nHeaterNumber]*10, nHeaterNumber); //Move the decimal point by 1
			END_IF
			IF (bAutoTuneSV[nHeaterNumber] <> bAutoTuneTV[nHeaterNumber]) THEN
				bAutoTuneTV[nHeaterNumber] := bAutoTuneSV[nHeaterNumber];
				sSendString := BOOL_TO_STRING_LHeaterON(nHeaterNumber,bAutoTuneTV[nHeaterNumber]);
			END_IF
			
			TimeWaitSend(IN:=TRUE, PT:=T#10MS);
			IF TimeWaitSend.Q THEN
				TimeWaitSend(IN:=FALSE);
				IF fbSend.Busy THEN
					fbSend(	SendString:= sSendString,
						TXbuffer:= TxBufferLH,
						Busy=> bSendBusy,
						Error=> );
					IF fbSend.Error <> COMERROR_NOERROR THEN
						eSendErrorID := fbSend.Error;
						bSendingOK := FALSE;
					ELSE
						eSendErrorID := COMERROR_NOERROR;
						bSendingOK := TRUE;
					END_IF
				END_IF
			END_IF

		END_FOR
		
	END_IF
	
	TimeWaitSend(IN:=bSendingEnable AND bSendingOK = FALSE, PT:=T#10MS);
	IF TimeWaitSend.Q OR fbSend.Busy THEN
		bSendingOK := TRUE;
		fbSend(
			SendString := sSendString,
			TXBuffer := TXBufferLH,
			Busy => bSendBusy,
			Error =>
			);
		IF fbSend.Error <> COMERROR_NOERROR THEN
			eSendErrorID := fbSend.Error;
			bSendingOK := FALSE;
		ELSE
			bSendingOK := TRUE;
			bSendingOK := TRUE;
		END_IF
	END_IF
	
	fbReceive(
		Prefix := '$02',
		Suffix:= '$0D$0A',
		Timeout:= T#1S,
		ReceivedString:= sReceivedString,
		RXbuffer:=RXbufferLH,
		StringReceived=> bStringReceived,
		Busy=> bReceiveBusy,
		Error=>
		);
	IF bStringReceived THEN
		bStringReceived := FALSE;
		bReceivedOK:= TRUE;
		
		IF nComMode =1 THEN
			nStrPosition := 11;			
			FOR nHeaterNumber := 1 TO 8 DO
				hStrReceivedPV := MID(STR:=sReceivedString, LEN:=4, POS:=nStrPosition);
				rTemperaturePV[nHeaterNumber] := (HEXSTR_TO_REAL_LHeaterPV(hStrReceivedPV))/10; //Move the decimal point by 1
				nStrPosition := nStrPosition + 5;
			END_FOR
		ELSE
			nStrPosition := 11;		
			FOR nHeaterNumber := 1 TO 8 DO
				hStrReceivedST := MID(STR:=sReceivedString, LEN:=4, POS:=nStrPosition);						
				IF hStrReceivedST = '0002' THEN
					isLineHeater_Run[nHeaterNumber] 	:= TRUE;
					isLineHeater_ATune[nHeaterNumber] 	:= FALSE;
					isLineHeater_Err[nHeaterNumber] 	:= FALSE;
				ELSIF hStrReceivedST = '0004' THEN
					isLineHeater_Run[nHeaterNumber] 	:= FALSE;
					isLineHeater_ATune[nHeaterNumber] 	:= TRUE;
					isLineHeater_Err[nHeaterNumber] 	:= FALSE;
				ELSIF hStrReceivedST = '0080' THEN
					isLineHeater_Run[nHeaterNumber] 	:= FALSE;
					isLineHeater_ATune[nHeaterNumber] 	:= FALSE;
					isLineHeater_Err[nHeaterNumber] 	:= TRUE;
				ELSE
					isLineHeater_Run[nHeaterNumber] 	:= FALSE;
					isLineHeater_ATune[nHeaterNumber] 	:= FALSE;
					isLineHeater_Err[nHeaterNumber] 	:= FALSE;
				END_IF
				nStrPosition := nStrPosition + 5;		
			END_FOR
		END_IF
	END_IF
	
	TimeWaitReceive(IN:=bReceivedOK,PT:=T#1S);
	TimeCycle(IN:=TRUE, PT:=T#2S);
	IF TimeWaitReceive.Q OR TimeCycle.Q THEN
		TimeWaitReceive(IN:= TRUE);
		TimeCycle(IN:= FALSE);
		bSendingEnable := FALSE;
	END_IF
END_IF

END_PROGRAM

// ---- POUs/P20_BackgroundCom.TcPOU
PROGRAM P20_BackgroundCom
VAR
END_VAR

(* background communication with the EL6031 terminal to *)
// Thermal Bath x 6
// Line Heat x 8
P21_Background_LineHeater();
P22_Background_ThermalBath();

END_PROGRAM
